// TIA Portal V17 export
// export: Created 2023-02-14T02:49:41.8106859Z, ExportSetting WithDefaults, DisplayName Totally Integrated Automation Portal, DisplayVersion V17, DisplayName TIA Portal Openness, DisplayVersion V17, DisplayName TIA Portal Teamcenter Gateway, DisplayVersion V17, DisplayName TIA Portal Version Control Interface, DisplayVersion V17, DisplayName SINAMICS Startdrive Advanced, DisplayVersion V17, DisplayName SINAMICS Startdrive G130, G150, S120, S150, SINAMICS MV, S210, DisplayVersion V17, DisplayName SINAMICS Startdrive G110M, G120, G120C, G120D, G120P, G115D, DisplayVersion V17, DisplayName STEP 7 Professional, DisplayVersion V17, DisplayName STEP 7 Safety, DisplayVersion V17, DisplayName WinCC Professional, DisplayVersion V17
DATA_BLOCK "T-10_Vinegar"   // DB369
VERSION : 0.1
// stored: AutoNumber false, DBAccessibleFromOPCUA true, DBAccessibleFromWebserver true, InstanceOfName BFT_Vinegar, InstanceOfType FB
"BFT_Vinegar"
   // VAR_INPUT
   //    IN_FBAV_Inload : Bool;
   //    IN_FBAV_Outlet : Bool;
   //    IN_FBAV_Transfer : Bool;
   //    IN_FBAV_CIP_Tank : Bool;
   //    IN_FBAV_CIP_Line : Bool;
   //    IN_FBP_Inload : Bool;
   //    IN_FBP_Inload_SP : Real;
   //    IN_FBP_Transfer : Bool;
   //    IN_FBP_Transfer_SP : Real;
   //    IN_FBP_CIP : Bool;
   //    IN_FBP_CIP_Sp : Real;
   //    IN_LT01 : Real;
   //    "LCS Start" : Bool;
   //    "LCS Stop" : Bool;
   //    "LCS EMS" : Bool;
   //    IN_Dose_Run : Bool;
   //    IN_Dose_Held : Bool;
   //    IN_Dose_Complete : Bool;
   //    IN_Dose_Valve_Cmd : Bool;
   //    IN_Dose_Pump_Cmd : Bool;
   //    IN_Dose_Pump_Sp : Real;
   //    IN_Dose_LineOK : Bool;
   //    "Inload Busy" : Bool;
   //    "CIP Pulse" : Bool;
   //    "CIP Supply ON" : Bool;
   //    "CIP Req OK" : Bool;
   //    "CIP Complete" : Bool;
   //    "CIP Busy" : Bool;
   // END_VAR
   // VAR_OUTPUT
   //    Out_AV_Inload : Bool;
   //    Out_AV_Outlet : Bool;
   //    Out_AV_Transfer : Bool;
   //    Out_AV_CIP_Tank : Bool;
   //    Out_AV_CIP_Line : Bool;
   //    Out_P_Inload : Bool;
   //    Out_P_Inload_Sp : Real;
   //    Out_P_Transfer : Bool;
   //    Out_P_Transfer_Sp : Real;
   //    Out_P_CIP : Bool;
   //    Out_P_CIP_Sp : Real;
   //    Out_CIP_Req : Bool;
   //    Out_CIP_LineOpen : Bool;
   // END_VAR
   // VAR
   //    Cmd : Struct
   //       Inload : Bool;
   //       Ready_for_Tranfer : Bool;
   //       CIP_Tank : Bool;
   //       CIP_Line : Bool;
   //    END_STRUCT;
   // END_VAR
   // VAR RETAIN
   //    Param : Struct
   //       SP_Level_LL : Real;
   //       SP_Level_ML : Real;
   //       SP_Level_HL : Real;
   //       SupplyPump_SP_Speed : Real;
   //       L_Hi_Lim : Real;
   //       L_Lo_Lim : Real;
   //       L_Hys : Real;
   //       FlushingTime : DInt;
   //       CIP_Trf_SP_Speed : Real;
   //       CIP_Ret_ON_SP : Real;
   //       CIP_Ret_OFF_SP : Real;
   //    END_STRUCT;
   // END_VAR
   // VAR
   //    State : Struct
   //       Tank_LL : Bool;
   //       Tank_ML : Bool;
   //       Tank_HL : Bool;
   //       Tank_inCIP : Bool;
   //       Tank_CIP_Enable : Bool;
   //       Line_inCIP : Bool;
   //       Line_CIP_Enable : Bool;
   //       CIP_Return_On : Bool;
   //       Inloading : Bool;
   //       Inload_Enable : Bool;
   //       Ready_For_Transfer : Bool;
   //       Ready_For_Transfer_Ena : Bool;
   //       Tank_Available : Bool;
   //       Transfer_On_Prog : Bool;
   //    END_STRUCT;
   //    alwaysON : Bool;
   //    L_Hys_Abs : Real;
   //    Hys_Level_HL : Real;
   //    Hys_Level_ML : Real;
   //    Hys_Level_LL : Real;
   //    r : Struct
   //       PosE1 : Bool;
   //       PosE2 : Bool;
   //       PosE3 : Bool;
   //       PosE4 : Bool;
   //       PosE5 : Bool;
   //       PosE6 : Bool;
   //       PosE7 : Bool;
   //       PosE8 : Bool;
   //       PosE9 : Bool;
   //       PosE10 : Bool;
   //       PosE11 : Bool;
   //       PosE12 : Bool;
   //       PosE13 : Bool;
   //       PosE14 : Bool;
   //       PosE15 : Bool;
   //       PosE16 : Bool;
   //       PosE17 : Bool;
   //       PosE18 : Bool;
   //       PosE19 : Bool;
   //       PosE20 : Bool;
   //       PosE21 : Bool;
   //       PosE22 : Bool;
   //       PosE23 : Bool;
   //       PosE24 : Bool;
   //       PosE25 : Bool;
   //       PosE26 : Bool;
   //       PosE27 : Bool;
   //       PosE28 : Bool;
   //       PosE29 : Bool;
   //       PosE30 : Bool;
   //       PosE31 : Bool;
   //       PosE32 : Bool;
   //    END_STRUCT;
   //    Actuator : Struct
   //       AV_Inload : Bool;
   //       AV_Outlet : Bool;
   //       AV_Transfer : Bool;
   //       AV_CIP_Tank : Bool;
   //       AV_CIP_Line : Bool;
   //       P_Transfer : Bool;
   //       P_Inload : Bool;
   //       P_CIP : Bool;
   //       LCS_OnOff : Bool;
   //    END_STRUCT;
   //    FlushingTim : TON_TIME;
   //    SPumpTim { S7_SetPoint := 'True'} : TON_TIME;
   //    AVinloadTim { S7_SetPoint := 'True'} : TON_TIME;
   //    Pump_TF_On_Time { S7_SetPoint := 'True'} : TON_TIME;
   // END_VAR
BEGIN
END_DATA_BLOCK
